// Mitsubishi GX Works2 project: VB Net to RS485   PLC: FX3U/FX3UC

PROGRAM MAIN
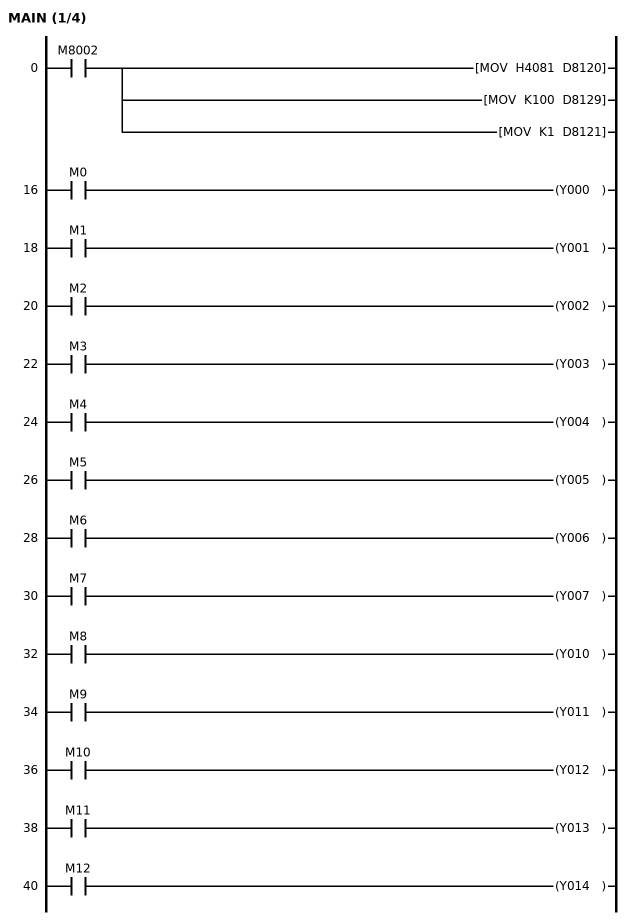
0     LD      M8002
      MOV     H4081 D8120
      MOV     K100 D8129
      MOV     K1 D8121
16    LD      M0
      OUT     Y000
18    LD      M1
      OUT     Y001
20    LD      M2
      OUT     Y002
22    LD      M3
      OUT     Y003
24    LD      M4
      OUT     Y004
26    LD      M5
      OUT     Y005
28    LD      M6
      OUT     Y006
30    LD      M7
      OUT     Y007
32    LD      M8
      OUT     Y010
34    LD      M9
      OUT     Y011
36    LD      M10
      OUT     Y012
38    LD      M11
      OUT     Y013
40    LD      M12
      OUT     Y014
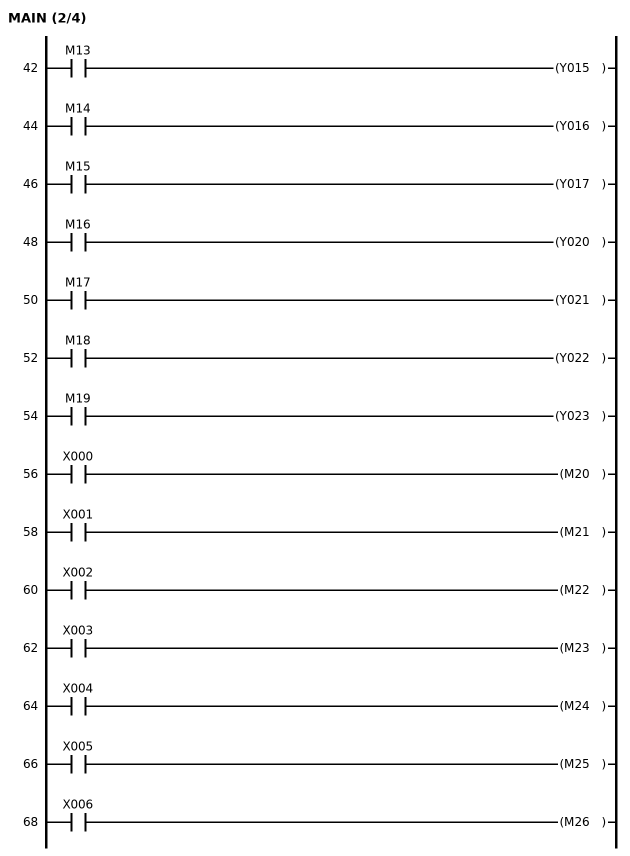
42    LD      M13
      OUT     Y015
44    LD      M14
      OUT     Y016
46    LD      M15
      OUT     Y017
48    LD      M16
      OUT     Y020
50    LD      M17
      OUT     Y021
52    LD      M18
      OUT     Y022
54    LD      M19
      OUT     Y023
56    LD      X000
      OUT     M20
58    LD      X001
      OUT     M21
60    LD      X002
      OUT     M22
62    LD      X003
      OUT     M23
64    LD      X004
      OUT     M24
66    LD      X005
      OUT     M25
68    LD      X006
      OUT     M26
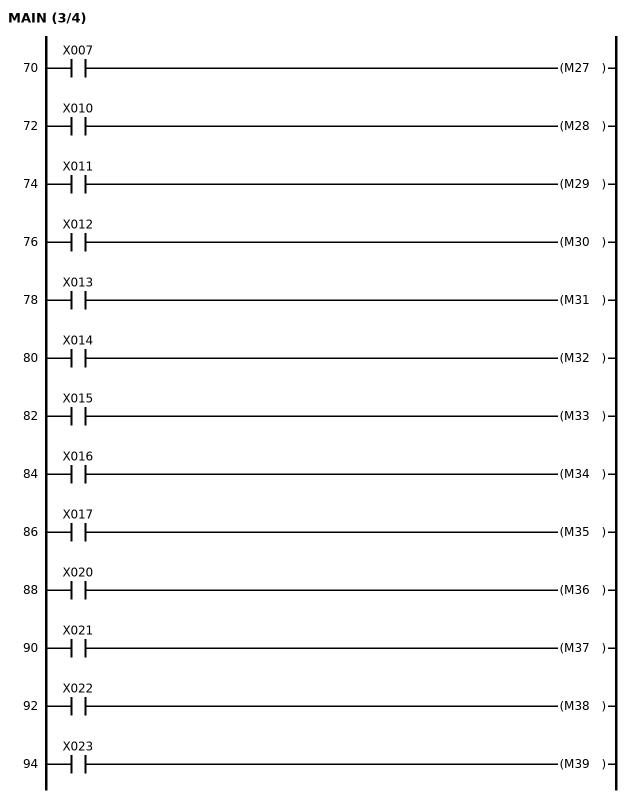
70    LD      X007
      OUT     M27
72    LD      X010
      OUT     M28
74    LD      X011
      OUT     M29
76    LD      X012
      OUT     M30
78    LD      X013
      OUT     M31
80    LD      X014
      OUT     M32
82    LD      X015
      OUT     M33
84    LD      X016
      OUT     M34
86    LD      X017
      OUT     M35
88    LD      X020
      OUT     M36
90    LD      X021
      OUT     M37
92    LD      X022
      OUT     M38
94    LD      X023
      OUT     M39
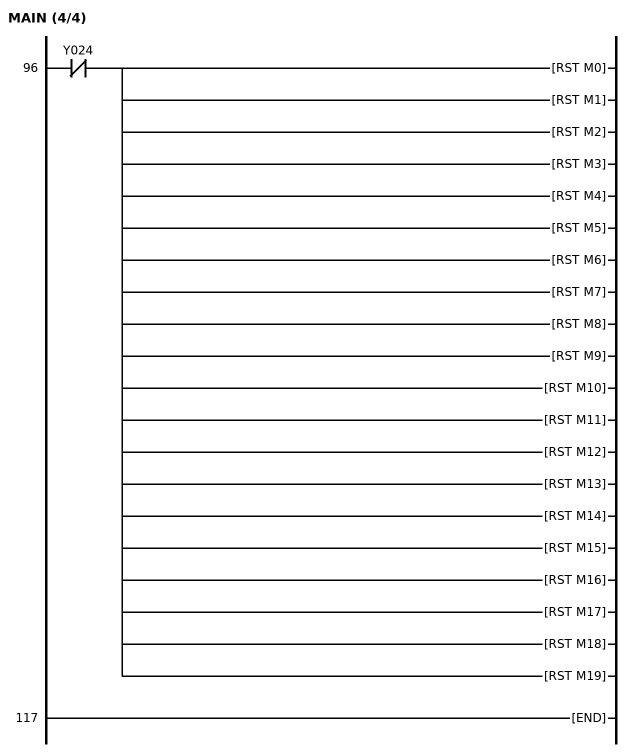
96    LDI     Y024
      RST     M0
      RST     M1
      RST     M2
      RST     M3
      RST     M4
      RST     M5
      RST     M6
      RST     M7
      RST     M8
      RST     M9
      RST     M10
      RST     M11
      RST     M12
      RST     M13
      RST     M14
      RST     M15
      RST     M16
      RST     M17
      RST     M18
      RST     M19
117   END
END_PROGRAM
